// TIA Portal V18 export
FUNCTION_BLOCK "Count_CycleTime_V3"   // FB3003, SCL
TITLE = Count_CycleTime
{ S7_Optimized_Access := 'TRUE' }
AUTHOR : STD
FAMILY : RCS
VERSION : 18.0
// 1.count
// 2.cycle time
// stored: AutoNumber false, IsIECCheckEnabled false, IsRetainMemResEnabled false, MemoryReserve 100, SetENOAutomatically false, UDAEnableTagReadback true
   VAR_INPUT
      iAlwaysOn : Bool;
      iProcessStart : Bool;
      iProcessComplete : Bool;
      iProcessResult : DInt;
   END_VAR
   VAR_IN_OUT
      ioCount : "RCS_SysCount_V1";
      ioTotalCycleTime : "RCS_SysCycleTime_V1";
      ioMachineCycleTime : "RCS_SysCycleTime_V1";
   END_VAR
   VAR
      sFlow : Struct
         pls : Array[0..15] of Bool;
         sDTStart : Date_And_Time;
         sDTRes : Date_And_Time;
         sDTOld : Date_And_Time;
         sDTRuntime : Date_And_Time;
         sDTRunning : Date_And_Time;
         sDTCurrent : Date_And_Time;
         Run_Minute : Int;
         Run_Hour : Int;
         Run_Day : Int;
         AutoRun_Minute : Int;
         AutoRun_Hour : Int;
         AutoRun_Day : Int;
      END_STRUCT;
   END_VAR
   VAR_TEMP
      tStart : Bool;
      tStop : Bool;
      tAutorunning : Bool;
      tpt : Int;
      tpRet : Int;
      tpResult : Time;
      tDint : DInt;
      tReal : Array[0..1] of Real;
   END_VAR
BEGIN
   (*############################################################
      RUHLAMAT SUZHOU ELEC.STD.
      Copyright (c) 2017. All rights reserved.    

      NAME OF FUNCTION BLOCK:         Count_CycleTimeV2.0
      VERSION NUMBER:                 V2.0
      COMPOSER:                       Ming.Jiang

      LAST CHANGE:                    13.April.2017
      Comment by Ming.Jiang 

      #RET_VALUE:


      #Alert Value:



      -----------------------------------------------------
      Date        Name      Version           Activity                                                                              

   ############################################################*)

   #tStart := #iProcessStart AND NOT #sFlow.pls[0];
   #sFlow.pls[0] := #iProcessStart;
   #tStop := #iProcessComplete AND NOT #sFlow.pls[1];
   #sFlow.pls[1] := #iProcessComplete;

   // IF #tStop THEN
   //     #tpRet := RD_SYS_T(#sFlow.sDTOld);
   // END_IF;

   //Machine Cycle time
   IF TRUE THEN
       IF #tStart THEN
           #tpRet := RD_SYS_T(#sFlow.sDTStart);
       END_IF;
       IF #tStop THEN

           //MachineTime
           #ioMachineCycleTime.No[21] := 0.0;
           #tpRet := RD_SYS_T(#sFlow.sDTRes);
           #tReal[0] := DINT_TO_REAL(TIME_TO_DINT(T_DIFF(IN1 := #sFlow.sDTRes, IN2 :=#sFlow.sDTStart )));
           #ioMachineCycleTime.No[0] :=  #tReal[0]/1000.0;

           //TotalTime
           #ioTotalCycleTime.No[21] := 0.0;
           #tReal[1] := DINT_TO_REAL(TIME_TO_DINT(T_DIFF(IN1 := #sFlow.sDTRes, IN2 := #sFlow.sDTOld)));
           #tpRet := RD_SYS_T(#sFlow.sDTOld);
           #ioTotalCycleTime.No[0] := #tReal[1]/1000.0;
           FOR #tpt := 20 TO 1 BY -1  DO
               //MachineTime
               #ioMachineCycleTime.No[#tpt] := #ioMachineCycleTime.No[#tpt - 1];
               #ioMachineCycleTime.No[21] := #ioMachineCycleTime.No[21] + #ioMachineCycleTime.No[#tpt];
               //totalCycleTime
               #ioTotalCycleTime.No[#tpt] := #ioTotalCycleTime.No[#tpt - 1];
               #ioTotalCycleTime.No[21] := #ioTotalCycleTime.No[21] + #ioTotalCycleTime.No[#tpt];
           END_FOR;
           //MachineTime
           #ioMachineCycleTime.No[21] := #ioMachineCycleTime.No[21] / 20.0;
           //totalCycleTime
           #ioTotalCycleTime.No[21] := #ioTotalCycleTime.No[21] / 20.0;

           //Count-------------------------------------------------------//
           IF #iProcessResult = 400 THEN
               #ioCount.OK[0] := #ioCount.OK[0] + 1;
               #ioCount.OKHolding := #ioCount.OKHolding + 1;
           END_IF;
           IF #iProcessResult >400 THEN
               #ioCount.NG[0] := #ioCount.NG[0] + 1;
               #ioCount.NGHolding:=#ioCount.NGHolding+1;
           END_IF;
           IF #iProcessResult >=400 THEN
               #ioCount.Total := #ioCount.Total + 1;
           END_IF;
           #ioCount.OKHolding := #ioCount.OKHolding + 1;

           CASE #iProcessResult OF
               401:  //NG1
                   #ioCount.NG[1] := #ioCount.NG[1] + 1;
               402:  //NG1uuuuuuuuuuuuuuuuuuuuuuuuuuuuuuuuuuuuuuuuuuuuuuuu
                   #ioCount.NG[2] := #ioCount.NG[2] + 1;
               403:  //NG1uuuuu
                   #ioCount.NG[3] := #ioCount.NG[3] + 1;
               404:  //NG1
                   #ioCount.NG[4] := #ioCount.NG[4] + 1;
               405:  //NG1
                   #ioCount.NG[5] := #ioCount.NG[5] + 1;
               406:  //NG1
                   #ioCount.NG[6] := #ioCount.NG[6] + 1;
               407:  //NG1
                   #ioCount.NG[7] := #ioCount.NG[7] + 1;
               408:  //NG1
                   #ioCount.NG[8] := #ioCount.NG[8] + 1;
               409:  //NG1
                   #ioCount.NG[9] := #ioCount.NG[9] + 1;

           END_CASE;
       END_IF;

   END_IF;
   //clear 
   IF #ioCount.ClearOK AND NOT #sFlow.pls[3] THEN
       #ioCount.OK[0] := 0;

   END_IF;
   #sFlow.pls[3] := #ioCount.ClearOK;
   IF #ioCount.ClearNG AND NOT #sFlow.pls[4] THEN
       FOR #tpt := 0 TO 9 DO
            #ioCount.NG[#tpt] := 0;
        END_FOR;
   END_IF;
   #sFlow.pls[4] := #ioCount.ClearNG;
   IF #ioCount.ClearTotal AND NOT #sFlow.pls[5] THEN
       #ioCount.Total := 0;

   END_IF;
   #sFlow.pls[5] := #ioCount.ClearTotal;
END_FUNCTION_BLOCK
